Fanuc KAREL source: WRITE_DICT_V.kl

PROGRAM T
%NOLOCKGROUP
VAR
 v0 : FILE
 v1 : STRING[40]
 v2 : INTEGER
 v3 : ARRAY[10] OF STRING[40]
 v4 : INTEGER
BEGIN
 WRITE_DICT_V(v0, v1, v2, v3, v4)
END T
